(* CoDeSys 2.3 export: GVL_CONST.EXP *)

(* Global variable list: GVL_CONST *)
VAR_GLOBAL CONSTANT
	iQtyD7Line: 		INT		:=25;		(*количество строк в расписании недельного таймера*)
	iMaxSelScrParam: 	INT		:=26;		(*максимальное количество строк на экране выбора параметра*)
	iStQty: 			INT		:=10;		(*количество шагов автоматической программы*)
	tUSDelay: 			TIME	:=t#1m;		(*задержка повторной подачи питания на УЗГ*)
	GlobalMaxRand: 		USINT	:=18;		(*количество рандомных значений и максимальное значение рандома*)
END_VAR
